ABB RAPID module: VSG_tooldata.sysx

MODULE VSG_tooldata(SYSMODULE)
    TASK PERS tooldata t_VSG_Servo   := [TRUE,[[0,0,114.2],[1,0,0,0]],[0.25,[8.2,11.7,52],[1,0,0,0],0.00021,0.00024,0.00009]];
    TASK PERS tooldata t_VSG_Vacuum1 := [TRUE, [[63.5, 18.5, 37.5], [0.70711, 0, 0.70711 ,0]], [0.25, [8.2, 11.7, 52.0], [1, 0, 0, 0], 0.00021, 0.00024, 0.00009]];
    TASK PERS tooldata t_VSG_Vacuum2 := [TRUE, [[-63.5, 18.5, 37.5], [0, -0.70711, 0, 0.70711]], [0.25, [8.2, 11.7, 52.0], [1, 0, 0, 0], 0.00021, 0.00024, 0.00009]];
ENDMODULE
